// TIA Portal V20 export
TYPE "typeSqlData"
TITLE = typeSqlData
// structure for SQL data received from SELECT command
   STRUCT
      tdsHeader { ExternalAccessible := 'False'; ExternalVisible := 'False'; ExternalWritable := 'False'} : "LSql_typePacketHeader";
      columnCount { ExternalAccessible := 'False'; ExternalVisible := 'False'; ExternalWritable := 'False'} : UInt;   // number of received columns
      columns { ExternalAccessible := 'False'; ExternalVisible := 'False'; ExternalWritable := 'False'} : Array[0.."LSQL_NUMBER_OF_COLUMNS_MAX"] of "LSql_typeColumn";
      rowDataStart { ExternalAccessible := 'False'; ExternalVisible := 'False'; ExternalWritable := 'False'} : UInt;   // start address byte of rowData in TDS telegram
      rowDataLength { ExternalAccessible := 'False'; ExternalVisible := 'False'; ExternalWritable := 'False'} : UDInt;   // area length of rowData in TDS telegram
      rowCount { ExternalAccessible := 'False'; ExternalVisible := 'False'; ExternalWritable := 'False'} : UDInt;   // number of rows
      rowOverflow { ExternalAccessible := 'False'; ExternalVisible := 'False'; ExternalWritable := 'False'} : Bool;   // true = more rows (RowCount) than available UDT tokenRows
      rows { ExternalAccessible := 'False'; ExternalVisible := 'False'; ExternalWritable := 'False'} : Array[0.."LSQL_NUMBER_OF_ROWS_MAX"] of "typeTokenRow";
      errorToken { ExternalAccessible := 'False'; ExternalVisible := 'False'; ExternalWritable := 'False'} : "LSql_typeErrorToken";
   END_STRUCT;
   // // tdsHeader."type" : type of TDS package (4 = Server Response)
   // // tdsHeader.status : status of the TDS package (1= last package, 0 = more packages follow)
   // // tdsHeader.length : length of the TDS response
   // // tdsHeader.spId : process id of the SQL server
   // // tdsHeader.packetID : id of one message for a paket
   // // tdsHeader.window : not used - should be ignored by user
END_TYPE
